INTERFACE I_ShakeMovement

PROPERTY P_Return : REFERENCE to ST_CommandReturn
GET
END_GET
END_PROPERTY

METHOD StartMovement
VAR_INPUT
	NumCycles		: UINT;
	Velo			: LREAL;
END_VAR
END_METHOD

END_INTERFACE

(* stored: Version 1.1.0.1, ProductVersion 3.1.4024.9
   Itf I_ShakeMovement: Id {f685737d-4101-48dd-8223-9d1e9c189bd8}
   Property P_Return: Id {3fae7c54-a3f7-4f58-8624-bf4b7f364047}
   Get Get: Id {a54ffea6-5cc7-4015-adba-c7c1637a9022}
   Method StartMovement: Id {4b3184dc-6ac8-40cf-993c-e9986ffe4194} *)
